FUNCTION_BLOCK TFCalcolaQuotaIngombroColonneLastre
VAR_INPUT
	QuotaY_ColonnaDX : LREAL; 		(* Quota della colonna a destra *)
	QuotaY_ColonnaSX : LREAL; 		(* Quota della colonna a destra *)
	QuotaAttualeAsse : LREAL; 		(* Quota attuale dell'asse Y*)
	QuotaDestinazioneAsse : LREAL; 	(* Quota Destinazione Asse Y*)
	IngombroOttimizzatoY_InTransito_Pos	: LREAL; (* Ingombro massimo della Y durante il ciclo in direzione POSITIVA *)
	IngombroOttimizzatoY_InTransito_Neg	: LREAL; (* Ingombro massimo della Y durante il ciclo in direzione NEGATIVA *)

	OffsetSicurezza_Y				: LREAL;  (* Offset sicurezza che si vuole mantenere dalle colonne *)
END_VAR
VAR_OUTPUT
	QuotaFuoriIngombro_Attuale_Y	: LREAL;
	QuotaFuoriIngombro_Destinazione_Y	: LREAL;
	//QuotaFuoriIngombro_Deposito_Y	: LREAL;
	Pinza_InIngombroColonne_Destinazione	: BOOL;
	Pinza_InIngombroColonne_Attuale			: BOOL;
END_VAR
VAR
	
END_VAR

(* Valutazione colonne in base al verso del pallettizzatore: verso stabilito guardando il pallettizzatore con la linea alle spalle *)
CASE VERSO_PALLETTIZZATORE OF
	PALLETTIZZATORE_DX:	// Colonna 6:DX, 5:SX
		(* Valuto la posizione attuale *)
		Pinza_InIngombroColonne_Attuale := FALSE;
		IF (QuotaAttualeAsse + IngombroOttimizzatoY_InTransito_Neg + OffsetSicurezza_Y <= QuotaY_ColonnaDX) THEN //Posizione Pinza - Metà ingombro - Offset sicurezza <= Ingombro colonna DX
			QuotaFuoriIngombro_Attuale_Y := QuotaY_ColonnaDX - IngombroOttimizzatoY_InTransito_Neg/2 - OffsetSicurezza_Y;
			Pinza_InIngombroColonne_Attuale := TRUE;
		END_IF
		IF (QuotaAttualeAsse - IngombroOttimizzatoY_InTransito_Pos - OffsetSicurezza_Y >= QuotaY_ColonnaSX) THEN //Posizione Pinza + Metà ingombro + Offset sicurezza >= Ingombro colonna SX
			QuotaFuoriIngombro_Attuale_Y := QuotaY_ColonnaSX + IngombroOttimizzatoY_InTransito_Pos/2 + OffsetSicurezza_Y;
			Pinza_InIngombroColonne_Attuale := TRUE;
		END_IF
		
		(* Valuto la posizione futura - Missione di Deposito/Prelievo *)
		Pinza_InIngombroColonne_Destinazione := FALSE;
		IF (QuotaDestinazioneAsse + IngombroOttimizzatoY_InTransito_Neg + OffsetSicurezza_Y <= QuotaY_ColonnaDX) THEN //Posizione Pinza - Metà ingombro - Offset sicurezza <= Ingombro colonna DX
			QuotaFuoriIngombro_Destinazione_Y := QuotaY_ColonnaDX - IngombroOttimizzatoY_InTransito_Neg - OffsetSicurezza_Y; 
			Pinza_InIngombroColonne_Destinazione := TRUE;
		END_IF
		IF (QuotaDestinazioneAsse - IngombroOttimizzatoY_InTransito_Pos - OffsetSicurezza_Y >= QuotaY_ColonnaSX) THEN //Posizione Pinza + Metà ingombro + Offset sicurezza >= Ingombro colonna SX
			QuotaFuoriIngombro_Destinazione_Y := QuotaY_ColonnaSX + IngombroOttimizzatoY_InTransito_Pos + OffsetSicurezza_Y;
			Pinza_InIngombroColonne_Destinazione := TRUE;
		END_IF
					
	PALLETTIZZATORE_SX: // Colonna 6:SX, 5:DX
		(* Valuto la posizione attuale *)
		Pinza_InIngombroColonne_Attuale := FALSE;
		IF (QuotaAttualeAsse + IngombroOttimizzatoY_InTransito_Pos + OffsetSicurezza_Y >= QuotaY_ColonnaDX) THEN //Posizione Pinza - Metà ingombro - Offset sicurezza <= Ingombro colonna 
			QuotaFuoriIngombro_Attuale_Y := QuotaY_ColonnaDX - IngombroOttimizzatoY_InTransito_Pos - OffsetSicurezza_Y;
			Pinza_InIngombroColonne_Attuale := TRUE;
		END_IF
		IF (QuotaAttualeAsse - IngombroOttimizzatoY_InTransito_Neg - OffsetSicurezza_Y <= QuotaY_ColonnaSX) THEN //Posizione Pinza + Metà ingombro + Offset sicurezza <= Ingombro colonna 
			QuotaFuoriIngombro_Attuale_Y := QuotaY_ColonnaSX + IngombroOttimizzatoY_InTransito_Neg + OffsetSicurezza_Y;
			Pinza_InIngombroColonne_Attuale := TRUE;
		END_IF
							
		(* Valuto la posizione futura - Missione di prelievo *)
		Pinza_InIngombroColonne_Destinazione := FALSE;
		IF (QuotaDestinazioneAsse + IngombroOttimizzatoY_InTransito_Pos + OffsetSicurezza_Y >= QuotaY_ColonnaDX) THEN //Posizione Pinza - Metà ingombro - Offset sicurezza <= Ingombro colonna 
			QuotaFuoriIngombro_Destinazione_Y := QuotaY_ColonnaDX - IngombroOttimizzatoY_InTransito_Pos - OffsetSicurezza_Y;
			Pinza_InIngombroColonne_Destinazione := TRUE;
		END_IF
		IF (QuotaDestinazioneAsse - IngombroOttimizzatoY_InTransito_Neg - OffsetSicurezza_Y <= QuotaY_ColonnaSX) THEN //Posizione Pinza + Metà ingombro + Offset sicurezza >= Ingombro colonna
			QuotaFuoriIngombro_Destinazione_Y := QuotaY_ColonnaSX + IngombroOttimizzatoY_InTransito_Neg + OffsetSicurezza_Y; 
			Pinza_InIngombroColonne_Destinazione := TRUE;
		END_IF

END_CASE

(* Nel caso in cui la pinza non sia in ingombro, fisso come fuori ingombro la quota attuale/ quota di destinazione dell'asse *)
IF NOT Pinza_InIngombroColonne_Attuale THEN
	QuotaFuoriIngombro_Attuale_Y := QuotaAttualeAsse;
END_IF
(* Nel caso in cui la pinza non sia in ingombro, fisso come fuori ingombro la quota di destinazione dell'asse *)
IF NOT Pinza_InIngombroColonne_Destinazione THEN
	QuotaFuoriIngombro_Destinazione_Y := QuotaAttualeAsse;
END_IF

END_FUNCTION_BLOCK

(* stored: Version 1.1.0.1, ProductVersion 3.1.4024.11
   POU TFCalcolaQuotaIngombroColonneLastre: Id {d5625752-e2c4-4910-a6dd-f27e993c65d4}, SpecialFunc None *)
